FUNCTION_BLOCK UDINT2REAL_2 (* Basic Function Block Type *)
  (* Standard: 61499-2 *)
  (* Version 0.0, 7/4/2026, Schneider Electric, Template *)
  PACKAGE SE.Nereda;
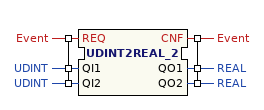
  EVENT_INPUT
    REQ WITH QI1, QI2; (* Normal Execution Request *)
  END_EVENT
  EVENT_OUTPUT
    CNF WITH QO1, QO2; (* Execution Confirmation *)
  END_EVENT
  VAR_INPUT
    QI1 : UDINT; (* Input event qualifier *)
    QI2 : UDINT;
  END_VAR
  VAR_OUTPUT
    QO1 : REAL; (* Output event qualifier *)
    QO2 : REAL;
  END_VAR
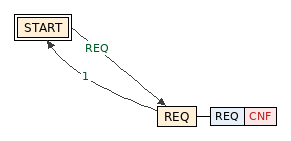
  EC_STATES
    START; (* Initial State *)
    REQ : REQ -> CNF; (* Normal execution *)
  END_STATES
  EC_TRANSITIONS
    START TO REQ := REQ;
    REQ TO START := 1;
  END_TRANSITIONS
  ALGORITHM REQ IN ST: (* Normally executed algorithm *)
;
QO1 := UDINT_TO_REAL(QI1);
QO2 := UDINT_TO_REAL(QI2);
  END_ALGORITHM
END_FUNCTION_BLOCK
